TYPE ST_ParseContext :
STRUCT
    stBuffer    	: ST_Span;
    stState     	: ST_ParserInternalState;
	pCurrentContext : POINTER TO FB_ParseContext; 	// The current context we are operating on
END_STRUCT
END_TYPE

(* stored: Version 1.1.0.1
   DUT ST_ParseContext: Id {95883e15-46b0-4bcb-bbdc-d8888725c7a3} *)
